// TwinCAT 3 PLC project EventVideoPlayback
// Title: Event Video Playback
// Company: Beckhoff Automation LLC
// ProjectVersion: 1.1.1
// ProgramVersion: 3.1.4026.19
// CompilerDefines: VISU_USEPROPERTYINFO
// libraries:
//   Tc2_Standard, * (Beckhoff Automation GmbH)
//   Tc2_System, * (Beckhoff Automation GmbH)
//   Tc2_Utilities, * (Beckhoff Automation GmbH)
//   Tc3_EventLogger, * (Beckhoff Automation GmbH)
//   Tc3_JsonXml, * (Beckhoff Automation GmbH)
//   Tc3_Vision, * (Beckhoff Automation GmbH)
// project tree:
//   / Parameters_EventVideoPlayback.TcGVL
//   Project Information/ F_GetCompany.TcPOU, F_GetTitle.TcPOU, F_GetVersion.TcPOU
//   VideoPlayback/ FB_ImageToVideo.TcPOU

// ---- Parameters_EventVideoPlayback.TcGVL
{attribute 'qualified_only'}
VAR_GLOBAL CONSTANT
	MAX_NUMBER_IMAGES_2_VIDEO : UDINT := 200;
	MAX_PERCENT_ROUTER_MEM_FOR_BUFFER : UDINT := 50;
	ADS_PORT_FOR_IMAGE_TO_VIDEO		  : UINT  := 26129;
	LARGE_ROUTER_MEMORY				  : UINT  := 4096;
END_VAR

// ---- Project Information/F_GetCompany.TcPOU
// This function has been automatically generated from the project information.
{attribute 'signature_flag' := '1073741824'}
{attribute 'TcGenerated'}
{attribute 'no-analysis'}
FUNCTION F_GetCompany : WSTRING
VAR_INPUT
	
END_VAR

F_GetCompany := "Beckhoff Automation LLC";

END_FUNCTION

// ---- Project Information/F_GetTitle.TcPOU
// This function has been automatically generated from the project information.
{attribute 'signature_flag' := '1073741824'}
{attribute 'TcGenerated'}
{attribute 'no-analysis'}
FUNCTION F_GetTitle : WSTRING
VAR_INPUT
	
END_VAR

F_GetTitle := "Event Video Playback";

END_FUNCTION

// ---- Project Information/F_GetVersion.TcPOU
// This function has been automatically generated from the project information.
{attribute 'signature_flag' := '1073741824'}
{attribute 'TcGenerated'}
{attribute 'no-analysis'}
FUNCTION F_GetVersion : ST_LibVersion
VAR_INPUT
	
END_VAR

F_GetVersion.iMajor := 1;
F_GetVersion.iMinor := 1;
F_GetVersion.iBuild := 1;
F_GetVersion.iRevision := 0;
F_GetVersion.sVersion := '1.1.1';
F_GetVersion.nFlags := 0;

END_FUNCTION

// ---- VideoPlayback/FB_ImageToVideo.TcPOU
FUNCTION_BLOCK FB_ImageToVideo EXTENDS FB_ListenerBase2
VAR_INPUT
END_VAR

VAR_OUTPUT
END_VAR

VAR
	//Base FB
	Error_FailedToWriteImagesToDisk : BOOL;
	_Busy							: BOOL := FALSE;
	_Error							: BOOL;
	_ErrorID						: UDINT;

	// Cyclic FB
	_InitComplete : BOOL;
	SequenceState : INT;

	// Reset
	_Reset				: BOOL;
	TriggerVideoCapture : BOOL;
	VideoCaptureState	: INT;

	//Interface

	// Ring Buffer information
	BufferImageRing		 : ARRAY[1..Parameters_EventVideoPlayback.MAX_NUMBER_IMAGES_2_VIDEO] OF ITcVnImage;
	BufferIndex			 : UINT := 1;
	CurrentBufferMax	 : UINT;
	WriteImageWaitResult : BOOL;
	ipImageToSave		 : ITcVnImage;
	WriteFileState		 : INT;
	sImageToSaveName	 : STRING;
	fbWriteImage		 : FB_VN_WriteImage;
	_fbEvent			 : REFERENCE TO FB_TcEvent;
	BufferHasRolledOver	 : BOOL := FALSE;

	// Video creation vars
	writeADS   : ADSWRITE;
	DoWrite	   : BOOL;
	JSONData   : T_MaxString;
	JsonWriter : FB_JsonSaxWriter;

	//Check connection to service
	writeADSConnection : ADSWRITE;

	//filename vars
	TimeDateStamp					: T_MaxString;
	GetTimeZone						: FB_GetTimeZoneInformation;
	TimeZoneInfo					: ST_TimeZoneInformation;
	SystemTimeToTzSpecificLocalTime : FB_SystemTimeToTzSpecificLocalTime;

	// Json vars to send to the C# app
	JsonFileName	: T_MaxString;
	JsonImageSource : T_MaxString;

	// Properties to build image
	_VideoOutputDirectory : STRING := 'C:\TcAlarmVideo';
	_FramesPerSecond	  : UINT   := 10; //Set to 10 so no divide by zero if not setup
	_CameraName			  : STRING := 'Camera1';
	_JSONAttribute		  : T_MaxString;
	_ReductionFactor	  : LREAL := 0.25;

	// Alarm data
	sJsonAttribute	 : STRING(10000);
	JSONFilter		 : FB_TcEventFilter;
	_Subscribe		 : BOOL := TRUE;
	_Unsubscribe	 : BOOL;
	_Subscribed		 : BOOL;
	MissedEventCount : UDINT;

	// Image count value
	ImageWriteCount : UINT;

	// Delay after alarm to wait then do work
	AfterEventDelay	  : TON;
	_TimeAfterEvent	  : TIME := T#3S;
	_TimeBeforeEvent  : TIME := T#7S;
	VideoCaptureAlarm : ARRAY[1..4] OF FB_TcAlarm;

	// Calculation of Video length variables
	VideoLengthCalculated					: LREAL;
	VideoAskedLength						: LREAL;
	Error_VideoConfigTooLongForBufferSize	: BOOL;
	Error_ImageBufferOrRouterMemoryTooSmall : BOOL;
	ImageMemCheckSize						: ULINT := 0;
	RouterMem								: FB_GetRouterStatusInfo;
	RouterInfo								: ST_TcRouterStatusInfo;
	NumberOfFramesPossibleByMemory			: ULINT;
	CheckConnection							: BYTE := 1;
	Check3rdParty_TON						: TON;
	Check3rdPartyRunning					: BOOL;
	DelayTON								: TON;
END_VAR

METHOD AddImage
VAR_INPUT
	ipImageIn : ITcVnImage;
END_VAR

VAR
	hrWD1					 : HRESULT;
	tStop1					 : DINT := 20000;
	tRest1					 : DINT;
	hr						 : HRESULT;
	///PixelFormat				 : TcVnPixelFormat;
	ImageInfo				 : TcVnImageInfo;
	ImagePixelFormatChannels : BYTE;
	ImageEffectivePixelSize	 : UINT;
	ImageInWidth			 : UDINT;
	ImageInHeight			 : UDINT;
	ImageSmallWidth			 : UDINT;
	ImageSmallHeight		 : UDINT;
END_VAR
IF NOT WriteImageWaitResult AND NOT _ERROR THEN
	hrWD1 := F_VN_StartRelWatchdog(tStop1, S_OK);

	// reduce the image if needed
	hr						 := F_VN_GetImageInfo(ipImage := ipImageIn, stImageInfo := ImageInfo, hrPrev := hr);
	ImagePixelFormatChannels := ImageInfo.stPixelFormat.nChannels;
	ImageEffectivePixelSize	 := ImageInfo.stPixelFormat.nElementSize;
	ImageInWidth			 := ImageInfo.nWidth;
	ImageInHeight			 := ImageInfo.nHeight;
	IF _ReductionFactor <> 1 THEN
		ImageSmallWidth	 := LREAL_TO_UDINT(UDINT_TO_LREAL(ImageInWidth) * _ReductionFactor);
		ImageSmallHeight := LREAL_TO_UDINT(UDINT_TO_LREAL(ImageInHeight) * _ReductionFactor);

		// Image Width and Height must be even for video conversion
		IF (ImageSmallWidth MOD 2) <> 0 THEN // Check if "Odd"
			ImageSmallWidth := ImageSmallWidth - 1;
		END_IF

		IF (ImageSmallHeight MOD 2) <> 0 THEN // Check if "Odd"
			ImageSmallHeight := ImageSmallHeight - 1;
		END_IF

		hr := F_VN_ResizeImage(ipImageIn,
							   BufferImageRing[BufferIndex],
							   ImageSmallWidth,
							   ImageSmallHeight,
							   1,
							   hr);
	ELSE
		hr := F_VN_CopyImage(ipImageIn, BufferImageRing[BufferIndex], hr);
	END_IF

	hrWD1		:= F_VN_StopWatchdog(hrWD1, tRest => tRest1);
	BufferIndex := BufferIndex + 1;
	IF BufferIndex > CurrentBufferMax THEN
		BufferHasRolledOver := TRUE;
		BufferIndex			:= 1;
	END_IF
END_IF
END_METHOD

PROPERTY Busy : BOOL
GET
Busy := _Busy;
END_GET
END_PROPERTY

PROPERTY CameraName : STRING
SET
_CameraName := CameraName;
END_SET
END_PROPERTY

METHOD PUBLIC CyclicLogic
VAR_INPUT
END_VAR

VAR
	hr				: HRESULT;
	tmpIndex		: UINT;
	systemTimeNow	: TIMESTRUCT;
	tmpString		: STRING;
	EventTimestamp1 : TimeStruct;
	EventTimestamp2 : TimeStruct;
	sDump			: STRING;
	TmpMemory		: ULINT;
END_VAR

VAR_INST
	x : UINT;
END_VAR
IF NOT _InitComplete THEN
	_InitComplete := Initialize();
	RETURN;
END_IF

// Call the Listener Execute
Execute();

// Subscribe to the event logger to messages with the JSON Attribute
IF _Subscribe THEN
	_Subscribe := FALSE;
	JSONFilter.Clear().JsonAttribute.Value.EqualTo(_JSONAttribute); // define all events (messages and alarms) from this eventclass   
	hr := Subscribe2(JSONFilter);									// subscribe to retrieve defined events
	IF SUCCEEDED(hr) THEN
		_Subscribed := TRUE;
	END_IF
END_IF

IF _Unsubscribe THEN
	_Unsubscribe := FALSE;
	hr			 := Unsubscribe();
	IF SUCCEEDED(hr) THEN
		_Subscribed := FALSE;
	END_IF
END_IF

// This is the state engine for when an alarm occurs that needs a video
CASE VideoCaptureState OF
	0:
		IF TriggerVideoCapture THEN
			_Busy			  := TRUE;
			x				  := 1;
			VideoCaptureState := 10;
		END_IF

	10: // wait for delay time to capture images after event
		IF AfterEventDelay.Q THEN
			VideoCaptureState := 15;
		END_IF

	15: // save images needed for video playback
		WriteImageWaitResult := TRUE;
		tmpIndex			 := BufferIndex + x - 1;
		IF tmpIndex > CurrentBufferMax THEN
			tmpIndex := tmpIndex - CurrentBufferMax;
		END_IF

		IF WriteImage(Index := x, BufferImageSaveNameIndex := TmpIndex) THEN
			x := x + 1;
		END_IF

		IF x > CurrentBufferMax THEN
			TriggerVideoCapture	 := FALSE;
			VideoCaptureState	 := 20;
			WriteImageWaitResult := FALSE;
		END_IF

	20: // Build string paths and names

		// Time is UTC and we need it in local time zone. 
		EventTimestamp1 := FILETIME64_TO_SYSTEMTIME(_fbevent.nTimestamp);
		SystemTimeToTzSpecificLocalTime(in := EventTimestamp1, tzInfo := TimeZoneInfo, out => EventTimestamp2);
		TimeDateStamp := SYSTEMTIME_TO_STRING(EventTimestamp2);
		FindAndReplaceChar(ADR(TimeDateStamp),
						   ':',
						   '-',
						   ADR(TimeDateStamp),
						   SIZEOF(TimeDateStamp));

		FindAndSplitChar(sSeparatorChar	  := '.',
						 pSrcString		  := ADR(TimeDateStamp),
						 pLeftString	  := ADR(TimeDateStamp),
						 nLeftSize		  := SIZEOF(TimeDateStamp),
						 pRightString	  := ADR(sDump),
						 nRightSize		  := SIZEOF(sDump),
						 bSearchFromRight := FALSE);

		// FileName string creation
		JsonFileName := CONCAT(_VideoOutputDirectory, '\');
		JsonFileName := CONCAT(JsonFileName, _CameraName);
		JsonFileName := CONCAT(JsonFileName, '\');
		JsonFileName := CONCAT(JsonFileName, TimeDateStamp);
		JsonFileName := CONCAT(JsonFileName, '.mp4');
		
		

		// image source string creation
		JsonImageSource	  := CONCAT(_VideoOutputDirectory, '\');
		JsonImageSource	  := CONCAT(JsonImageSource, _CameraName);
		JsonImageSource	  := CONCAT(JsonImageSource, '\');
		JsonImageSource	  := CONCAT(JsonImageSource, 'images');
		VideoCaptureState := 30;
		

	30: // setup JSON pairs
		MEMSET(ADR(JSONData), 0, SIZEOF(JSONData));
		JsonWriter.ResetDocument();
		JsonWriter.StartObject();
		JsonWriter.AddKeyString('ImagePathSource', JsonImageSource);
		JsonWriter.AddKeyString('VideoFilename', JsonFileName);
		JsonWriter.AddKeyNumber('VideoFPS', _FramesPerSecond);
		JsonWriter.EndObject();
		JSONData		  := JsonWriter.GetDocument();
		VideoCaptureState := 40;
		

	40: // write JSON data
		DoWrite			  := TRUE;
		VideoCaptureState := 45;

	45:
		IF writeADS.BUSY AND NOT writeADS.ERR THEN
			VideoCaptureState := 50;
		ELSIF writeADS.ERR THEN
			_ErrorID		  := writeADS.ERRID;
			VideoCaptureState := 999;
		END_IF

	50: // wait for write to be done
		IF NOT writeADS.BUSY AND NOT writeADS.ERR THEN
			DoWrite			  := FALSE;
			VideoCaptureState := 60;
		ELSIF writeADS.ERR THEN
			_ErrorID		  := writeADS.ERRID;
			VideoCaptureState := 999;
		END_IF

	60: // extra scan
		VideoCaptureAlarm[E_VideoAlarm.Camera1Alarm].Clear(0, 0);
		_Busy			  := FALSE;
		VideoCaptureState := 0;

	999: // error handling
		VideoCaptureAlarm[E_VideoAlarm.Camera1Alarm].Clear(0, 0);
		VideoCaptureAlarm[E_VideoAlarm.ImageToVideoService].Raise(0);
		DoWrite			  := FALSE;
		_Busy			  := FALSE;
		_Error			  := TRUE;
		VideoCaptureState := 1000;

	1000:
		IF _Reset OR NOT VideoCaptureAlarm[E_VideoAlarm.ImageToVideoService].bRaised THEN
			_Error			  := FALSE;
			_ErrorID		  := 0;
			VideoCaptureState := 0;
			_Reset			  := FALSE;
		END_IF
END_CASE

writeADS(NETID	 := '',
		 PORT	 := Parameters_EventVideoPlayback.ADS_PORT_FOR_IMAGE_TO_VIDEO,
		 IDXGRP	 := 1,
		 IDXOFFS := 1,
		 WRITE	 := DoWrite,
		 LEN	 := TO_UDINT(LEN(JSONData)),
		 SRCADDR := ADR(JSONData),
		 TMOUT	 := T#10S);

AfterEventDelay(IN := VideoCaptureState = 10, PT := _TimeAfterEvent);

(* Calculations for checking the video FPS, TimeBefore + TimeAfter, And Parameter.Maxbuffer size while related to image size
	The parameters that can be adjusted
		1. FramesPerSecond
		2. Time Before Event
		3. Time Afeter Event
		4. MAX Number of Frames
		5. Reduction Factor
		
	Fixed Parameters
		1. The memmory - 50% of router memory (Parameter_Vision.MAX_PERCENT_ROUTER_MEM_FOR_BUFFER in %)	
*)

// Monitor the actual needed buffer size
CurrentBufferMax := TO_UINT((TO_LREAL(_TimeAfterEvent) + TO_LREAL(_TimeBeforeEvent)) / 1000.0 * TO_LREAL(_FramesPerSecond));
IF CurrentBufferMax > Parameters_EventVideoPlayback.MAX_NUMBER_IMAGES_2_VIDEO THEN
	CurrentBufferMax := TO_UINT(Parameters_EventVideoPlayback.MAX_NUMBER_IMAGES_2_VIDEO);
END_IF

// Calculated Video length from parameters
VideoLengthCalculated := CurrentBufferMax * 1000 / _FramesPerSecond;
VideoAskedLength	  := TO_LREAL(_TimeAfterEvent + _TimeBeforeEvent);
IF VideoAskedLength > VideoLengthCalculated THEN
	Error_VideoConfigTooLongForBufferSize := TRUE;
ELSE
	Error_VideoConfigTooLongForBufferSize := FALSE;
END_IF

(* Check to see if enough memory for what is expected
   Get the index to last picture taken*)
tmpIndex := BufferIndex - 1;
IF tmpIndex < 1 THEN
	tmpIndex := CurrentBufferMax;
END_IF

// Get Image size
F_VN_ExportImageSize(ipImage := BufferImageRing[tmpIndex], ImageMemCheckSize, S_OK);
IF ImageMemCheckSize > 0 THEN
	IF RouterInfo.maxMem = 0 THEN										  // Larger than 4095MB
		TmpMemory := TO_ULINT(Parameters_EventVideoPlayback.LARGE_ROUTER_MEMORY) * 1024 * 1024; //Check to see if user put in a value
	ELSE
		TmpMemory := RouterInfo.maxMem;
	END_IF

	NumberOfFramesPossibleByMemory := TO_ULINT(TO_LREAL(TmpMemory) * TO_LREAL(Parameters_EventVideoPlayback.MAX_PERCENT_ROUTER_MEM_FOR_BUFFER) / 100.0 / TO_LREAL(ImageMemCheckSize));
END_IF

// Is the size of the buffer Larger than that based on parameters than is given
IF CurrentBufferMax > NumberOfFramesPossibleByMemory AND ImageMemCheckSize > 0 THEN
	Error_ImageBufferOrRouterMemoryTooSmall := TRUE;
ELSE
	Error_ImageBufferOrRouterMemoryTooSmall := FALSE;
END_IF

// Set alarm if out of range for configuration
IF Error_VideoConfigTooLongForBufferSize THEN
	_Error := TRUE;
	VideoCaptureAlarm[E_VideoAlarm.VideoConfigTooLongForBufferSize].Raise();
END_IF

IF Error_ImageBufferOrRouterMemoryTooSmall THEN
	_Error := TRUE;
	VideoCaptureAlarm[E_VideoAlarm.RouterMemoryTooSmall].Raise();
END_IF

// Check if 3rd party app is connected to ADS 
Check3rdParty_TON(IN := VideoCaptureAlarm[E_VideoAlarm.ImageToVideoService].bRaised AND NOT Check3rdPartyRunning, PT := T#5S);
IF VideoCaptureAlarm[E_VideoAlarm.ImageToVideoService].bRaised AND (Check3rdParty_TON.Q OR Check3rdPartyRunning) THEN
	Check3rdPartyRunning := TRUE;

	// Do an ADS write to C# App to see if it is running
	writeADSConnection(PORT	   := Parameters_EventVideoPlayback.ADS_PORT_FOR_IMAGE_TO_VIDEO,
					   IDXGRP  := 10,
					   IDXOFFS := 10,
					   LEN	   := SIZEOF(CheckConnection),
					   SRCADDR := ADR(CheckConnection),
					   WRITE   := TRUE,
					   TMOUT   := T#3S);

	IF NOT writeADSConnection.BUSY THEN
		writeADSConnection(WRITE := FALSE);
		IF NOT writeADSConnection.ERR THEN
			VideoCaptureAlarm[E_VideoAlarm.ImageToVideoService].Clear(0, 0);
			_Error	 := FALSE;
			_ErrorID := 0;
		END_IF

		Check3rdPartyRunning := FALSE;
	END_IF
END_IF

// If Reset then clear the alarm
IF _Reset THEN
	IF VideoCaptureAlarm[E_VideoAlarm.Camera1Alarm].bRaised THEN
		VideoCaptureAlarm[E_VideoAlarm.Camera1Alarm].Clear(0,0);
	END_IF
	_Reset := FALSE;
END_IF
END_METHOD

PROPERTY Error : BOOL
GET
Error := _Error;
END_GET
END_PROPERTY

PROPERTY ErrorID : UDINT
GET
ErrorID := _ErrorID;
END_GET
END_PROPERTY

PROPERTY FramesPerSecond : UINT
SET
_FramesPerSecond := FramesPerSecond;
END_SET
END_PROPERTY

PROPERTY InitComplete : BOOL
GET
InitComplete := _InitComplete;
END_GET
END_PROPERTY

METHOD Initialize : BOOL
VAR_INPUT
END_VAR
CASE SequenceState OF
	// Get the Timezone
	0:
		GetTimeZone(sNetID	 := '',
					bExecute := TRUE,
					tTimeout := T#5S,
					tzInfo	 => TimeZoneInfo);

		IF NOT GetTimeZone.bBusy AND NOT GetTimeZone.bError THEN
			GetTimeZone(sNetID := '', bExecute := FALSE);
			SequenceState := 10;
		ELSIF GetTimeZone.bError THEN
			_Error		  := TRUE;
			_ErrorID	  := 16#FFFFFFFF;
			SequenceState := 10;
		END_IF

	// Get the router memory
	10:
		RouterMem(sNetId   := '',
				  bExecute := TRUE,
				  tTimeout := T#3S,
				  bBusy	   =>,
				  bError   =>,
				  nErrID   =>,
				  info	   => RouterInfo);

		IF NOT RouterMem.bBusy THEN
			RouterMem(sNetId := '', bExecute := FALSE);
			SequenceState := 20;
		END_IF

	// Create alarms
	20:
		_JSONAttribute := CONCAT(STR1 := '{CreateVid: 1, CameraName: "', STR2 := _CameraName);
		_JSONAttribute := CONCAT(STR1 := _JSONAttribute, STR2 := '"}',);
		VideoCaptureAlarm[E_VideoAlarm.Camera1Alarm].CreateEx(stEventEntry := TC_EVENTS.VideoAlarm.Camera1Alarm, bWithConfirmation := FALSE, ipSourceInfo := 0);
		VideoCaptureAlarm[E_VideoAlarm.Camera1Alarm].SetJsonAttribute(sJsonAttribute := _JSONAttribute);
		VideoCaptureAlarm[E_VideoAlarm.Camera1Alarm].ipArguments.AddString(value := _CameraName);
		VideoCaptureAlarm[E_VideoAlarm.ImageToVideoService].CreateEx(stEventEntry := TC_EVENTS.VideoAlarm.ImageToVideoService, bWithConfirmation := FALSE, ipSourceInfo := 0);
		VideoCaptureAlarm[E_VideoAlarm.RouterMemoryTooSmall].CreateEx(stEventEntry := TC_EVENTS.VideoAlarm.RouterMemoryTooSmall, bWithConfirmation := FALSE, ipSourceInfo := 0);
		VideoCaptureAlarm[E_VideoAlarm.VideoConfigTooLongForBufferSize].CreateEx(stEventEntry := TC_EVENTS.VideoAlarm.VideoConfigTooLongForBufferSize, bWithConfirmation := FALSE, ipSourceInfo := 0);
		SequenceState := 30;

	30: // This delay is to make sure we can talk to the ADS server correctly and not fail. Timing tested at 10s
		IF DelayTON.Q THEN
			SequenceState := 35;
		END_IF

	35:
		// Do an ADS write to C# App to see if it is running
		writeADSConnection(NETID   := '',
						   PORT	   := Parameters_EventVideoPlayback.ADS_PORT_FOR_IMAGE_TO_VIDEO,
						   IDXGRP  := 10,
						   IDXOFFS := 10,
						   LEN	   := SIZEOF(CheckConnection),
						   SRCADDR := ADR(CheckConnection),
						   WRITE   := TRUE,
						   TMOUT   := T#10S);

		IF NOT writeADSConnection.BUSY THEN
			writeADSConnection(WRITE := FALSE);
			IF writeADSConnection.ERR THEN
				VideoCaptureAlarm[E_VideoAlarm.ImageToVideoService].Raise(0);
				_Error	 := TRUE;
				_ErrorID := writeADSConnection.ERRID;
			END_IF

			SequenceState := 40;
		END_IF

	40:
		Initialize := TRUE;
END_CASE

DelayTON(IN := SequenceState = 30, PT := T#3S);
END_METHOD

PROPERTY IsImageBufferOrRouterMemoryTooSmall : bool
GET
IsImageBufferOrRouterMemoryTooSmall := Error_ImageBufferOrRouterMemoryTooSmall;
END_GET
END_PROPERTY

PROPERTY IsTooLongForBufferFPS : bool
GET
IsTooLongForBufferFPS := Error_VideoConfigTooLongForBufferSize;
END_GET
END_PROPERTY

PROPERTY JsonAttribute : T_MaxString
SET
_JSONAttribute := JsonAttribute;
END_SET
END_PROPERTY

METHOD OnAlarmRaised : HRESULT
VAR_INPUT
	fbEvent : REFERENCE TO FB_TcEvent;
END_VAR

VAR
	hr : HRESULT;
END_VAR
// This is where we actually do the work
IF NOT TriggerVideoCapture  AND BufferHasRolledOver THEN
	TriggerVideoCapture := TRUE;
	ImageWriteCount		:= 1;
	hr					:= fbEvent.GetJsonAttribute(sJsonAttribute, SIZEOF(sJsonAttribute));
	_fbEvent			REF= fbevent;
ELSE
	MissedEventCount := MissedEventCount + 1;
END_IF

OnAlarmRaised := S_OK;
END_METHOD

PROPERTY ReductionFactor : LREAL
SET
_ReductionFactor := ReductionFactor;
END_SET
END_PROPERTY

METHOD Reset
VAR_INPUT
END_VAR
IF VideoCaptureAlarm[E_VideoAlarm.RouterMemoryTooSmall].bRaised THEN
	VideoCaptureAlarm[E_VideoAlarm.RouterMemoryTooSmall].Clear(0,0);	
END_IF
IF VideoCaptureAlarm[E_VideoAlarm.VideoConfigTooLongForBufferSize].bRaised THEN
	VideoCaptureAlarm[E_VideoAlarm.VideoConfigTooLongForBufferSize].Clear(0,0);	
END_IF
_Error := FALSE;
_ErrorID := 0;
_Reset := TRUE;
END_METHOD

PROPERTY SubscribedEvents : BOOL
GET
SubscribedEvents := _Subscribed;
END_GET
END_PROPERTY

PROPERTY SubscribeEvents : BOOL
SET
_Subscribe := SubscribeEvents;
END_SET
END_PROPERTY

PROPERTY TimeAfterEvent : TIME
SET
_TimeAfterEvent := TimeAfterEvent;
END_SET
END_PROPERTY

PROPERTY TimeBeforeEvent : TIME
SET
_TimeBeforeEvent := TimeBeforeEvent;
END_SET
END_PROPERTY

METHOD PUBLIC TriggerAlarmForVideoCapture
VAR_INPUT
	LogEntryName : STRING;
END_VAR
IF NOT VideoCaptureAlarm[E_VideoAlarm.Camera1Alarm].bRaised AND BufferHasRolledOver THEN
	VideoCaptureAlarm[E_VideoAlarm.Camera1Alarm].ipArguments.Clear().AddString(LogEntryName).AddString(_CameraName);
	VideoCaptureAlarm[E_VideoAlarm.Camera1Alarm].Raise(0);
END_IF
END_METHOD

PROPERTY UnsubscribeEvents : BOOL
SET
_Unsubscribe := UnsubscribeEvents;
END_SET
END_PROPERTY

PROPERTY VideoOutputDirectory : STRING
SET
_VideoOutputDirectory := VideoOutputDirectory;
END_SET
END_PROPERTY

METHOD WriteImage : BOOL
VAR_INPUT
	BufferImageSaveNameIndex : UINT;
	Index					 : UINT;
END_VAR

VAR
	SysTimeAtImageSave : ULINT;
END_VAR
CASE WriteFileState OF
	0:
		sImageToSaveName := CONCAT(STR1 := _VideoOutputDirectory, '\');
		sImageToSaveName := CONCAT(STR1 := sImageToSaveName, _CameraName);
		sImageToSaveName := CONCAT(STR1 := sImageToSaveName, '\Images\Image');
		CASE Index OF // Add leading zeros to index number of image name
			0..9:
				sImageToSaveName := CONCAT(sImageToSaveName, '000');
				sImageToSaveName := CONCAT(sImageToSaveName, TO_STRING(Index));

			10..99:
				sImageToSaveName := CONCAT(sImageToSaveName, '00');
				sImageToSaveName := CONCAT(sImageToSaveName, TO_STRING(Index));

			100..999:
				sImageToSaveName := CONCAT(sImageToSaveName, '0');
				sImageToSaveName := CONCAT(sImageToSaveName, TO_STRING(Index));

		ELSE
			sImageToSaveName := CONCAT(sImageToSaveName, TO_STRING(Index));
		END_CASE;

		sImageToSaveName := CONCAT(sImageToSaveName, '.png');
		ipImageToSave	 := BufferImageRing[BufferImageSaveNameIndex];

		// Copy write image here
		fbWriteImage(ipImage   := ipImageToSave,
					 sFilePath := sImageToSaveName,
					 nTimeout  := T#500MS,
					 bWrite	   := TRUE);

		WriteFileState := 10;

	10:
		// sFilePath must contain the full path, image name and type
		fbWriteImage(sFilePath := '', bWrite := FALSE); // This updates the Busy
		IF NOT fbWriteImage.bBusy AND NOT fbWriteImage.bError THEN
			fbWriteImage(sFilePath := sImageToSaveName, bWrite := FALSE);
			WriteFileState		:= 0;
			Error_FailedToWriteImagesToDisk := FALSE;
			WriteImage			:= TRUE;
		ELSIF fbWriteImage.bError THEN
			fbWriteImage(sFilePath := sImageToSaveName, bWrite := FALSE);

			// Failure to write to disk
			Error_FailedToWriteImagesToDisk := TRUE;
			WriteFileState		:= 0;
		END_IF

ELSE
	WriteFileState := 0;
END_CASE
END_METHOD

END_FUNCTION_BLOCK
